TYPE ST_EXECUTION_TABLE :
STRUCT
	ActionType:E_ACTIONTYPE;
	X:LREAL;
	Y:LREAL;
	I:LREAL;
	J:LREAL;
	Clockwise:BOOL;
END_STRUCT
END_TYPE

(* stored: Version 1.1.0.1, ProductVersion 3.1.4024.10
   DUT ST_EXECUTION_TABLE: Id {c6c0cd99-40c6-4175-b75f-46fdd51d7e37} *)
